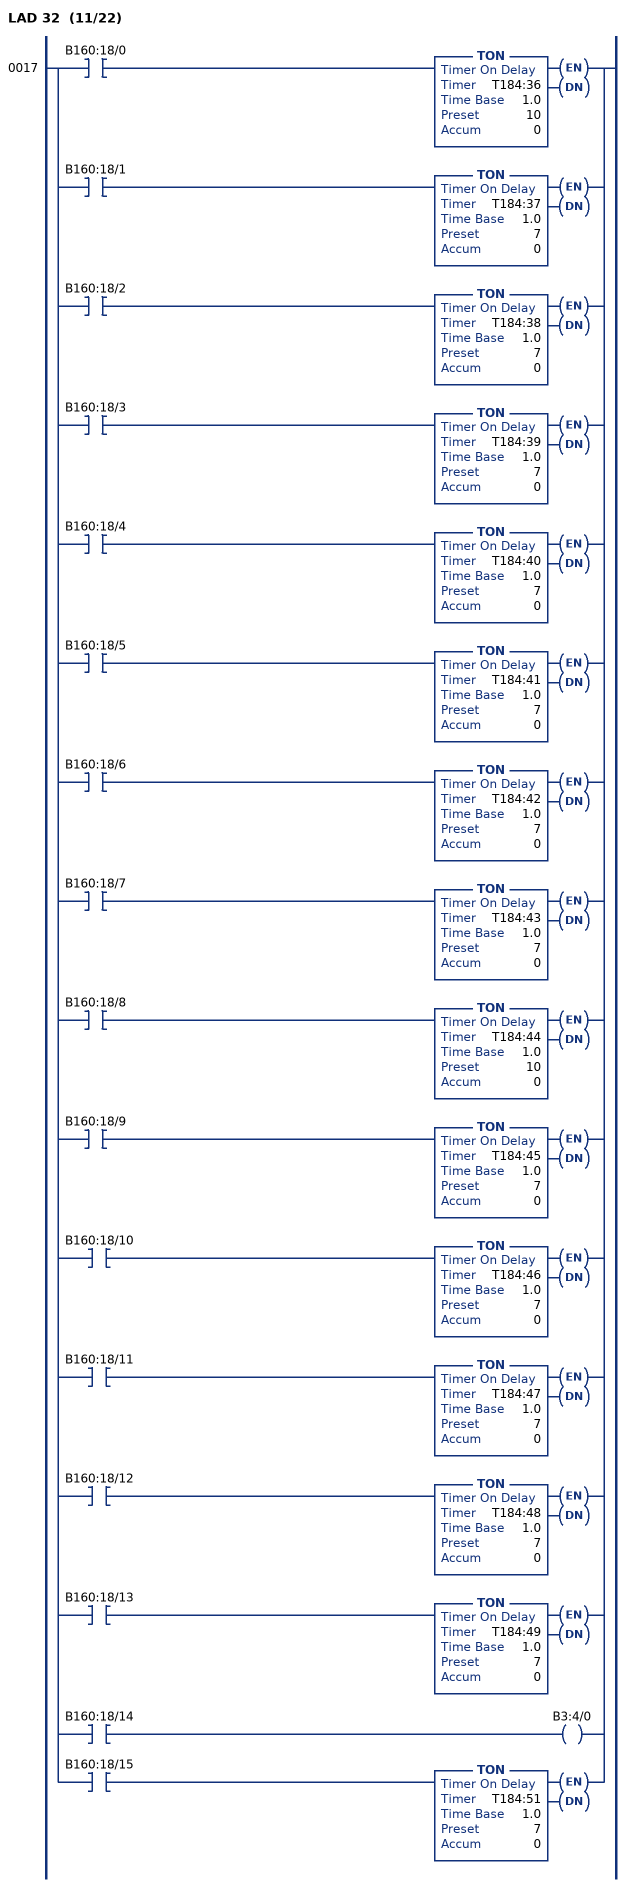
% Rung: 17 %
SOR BST XIC B160:18/0 TON T184:36 1.0 10 0 NXB XIC B160:18/1 TON T184:37 1.0 7 0 NXB XIC B160:18/2 TON T184:38 1.0 7 0 NXB XIC B160:18/3 TON T184:39 1.0 7 0 NXB XIC B160:18/4 TON T184:40 1.0 7 0 NXB XIC B160:18/5 TON T184:41 1.0 7 0 NXB XIC B160:18/6 TON T184:42 1.0 7 0 NXB XIC B160:18/7 TON T184:43 1.0 7 0 NXB XIC B160:18/8 TON T184:44 1.0 10 0 NXB XIC B160:18/9 TON T184:45 1.0 7 0 NXB XIC B160:18/10 TON T184:46 1.0 7 0 NXB XIC B160:18/11 TON T184:47 1.0 7 0 NXB XIC B160:18/12 TON T184:48 1.0 7 0 NXB XIC B160:18/13 TON T184:49 1.0 7 0 NXB XIC B160:18/14 OTE B3:4/0 NXB XIC B160:18/15 TON T184:51 1.0 7 0 BND EOR

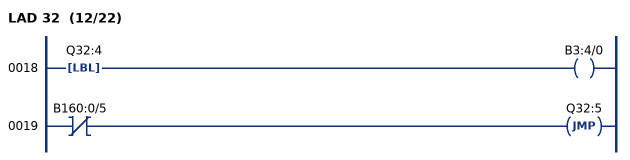
% Rung: 18 %
SOR LBL Q32:4 OTE B3:4/0 EOR
% Rung: 19 %
SOR XIO B160:0/5 JMP Q32:5 EOR

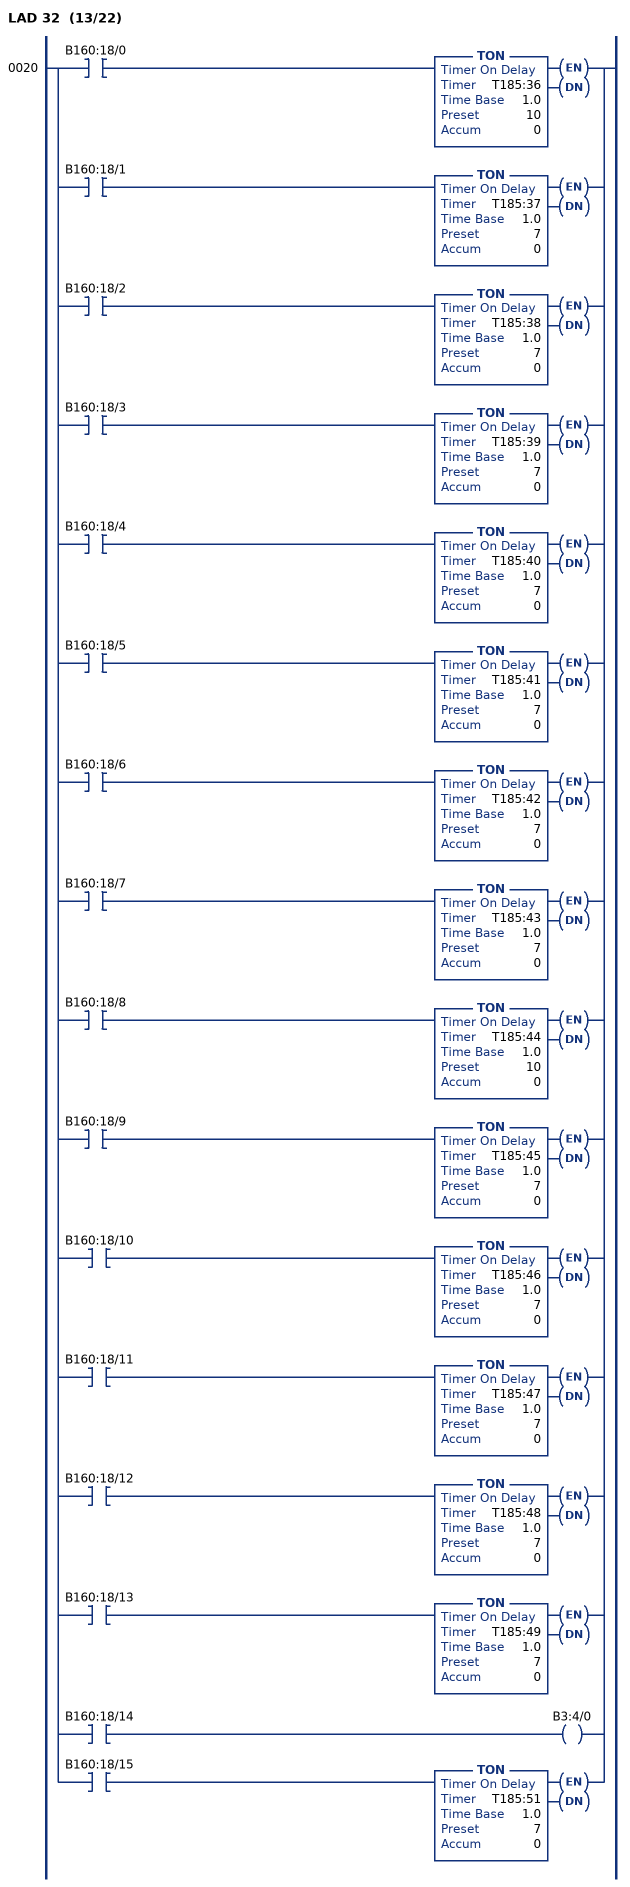
% Rung: 20 %
SOR BST XIC B160:18/0 TON T185:36 1.0 10 0 NXB XIC B160:18/1 TON T185:37 1.0 7 0 NXB XIC B160:18/2 TON T185:38 1.0 7 0 NXB XIC B160:18/3 TON T185:39 1.0 7 0 NXB XIC B160:18/4 TON T185:40 1.0 7 0 NXB XIC B160:18/5 TON T185:41 1.0 7 0 NXB XIC B160:18/6 TON T185:42 1.0 7 0 NXB XIC B160:18/7 TON T185:43 1.0 7 0 NXB XIC B160:18/8 TON T185:44 1.0 10 0 NXB XIC B160:18/9 TON T185:45 1.0 7 0 NXB XIC B160:18/10 TON T185:46 1.0 7 0 NXB XIC B160:18/11 TON T185:47 1.0 7 0 NXB XIC B160:18/12 TON T185:48 1.0 7 0 NXB XIC B160:18/13 TON T185:49 1.0 7 0 NXB XIC B160:18/14 OTE B3:4/0 NXB XIC B160:18/15 TON T185:51 1.0 7 0 BND EOR

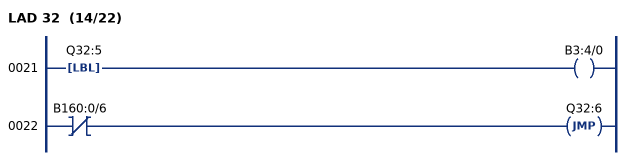
% Rung: 21 %
SOR LBL Q32:5 OTE B3:4/0 EOR
% Rung: 22 %
SOR XIO B160:0/6 JMP Q32:6 EOR

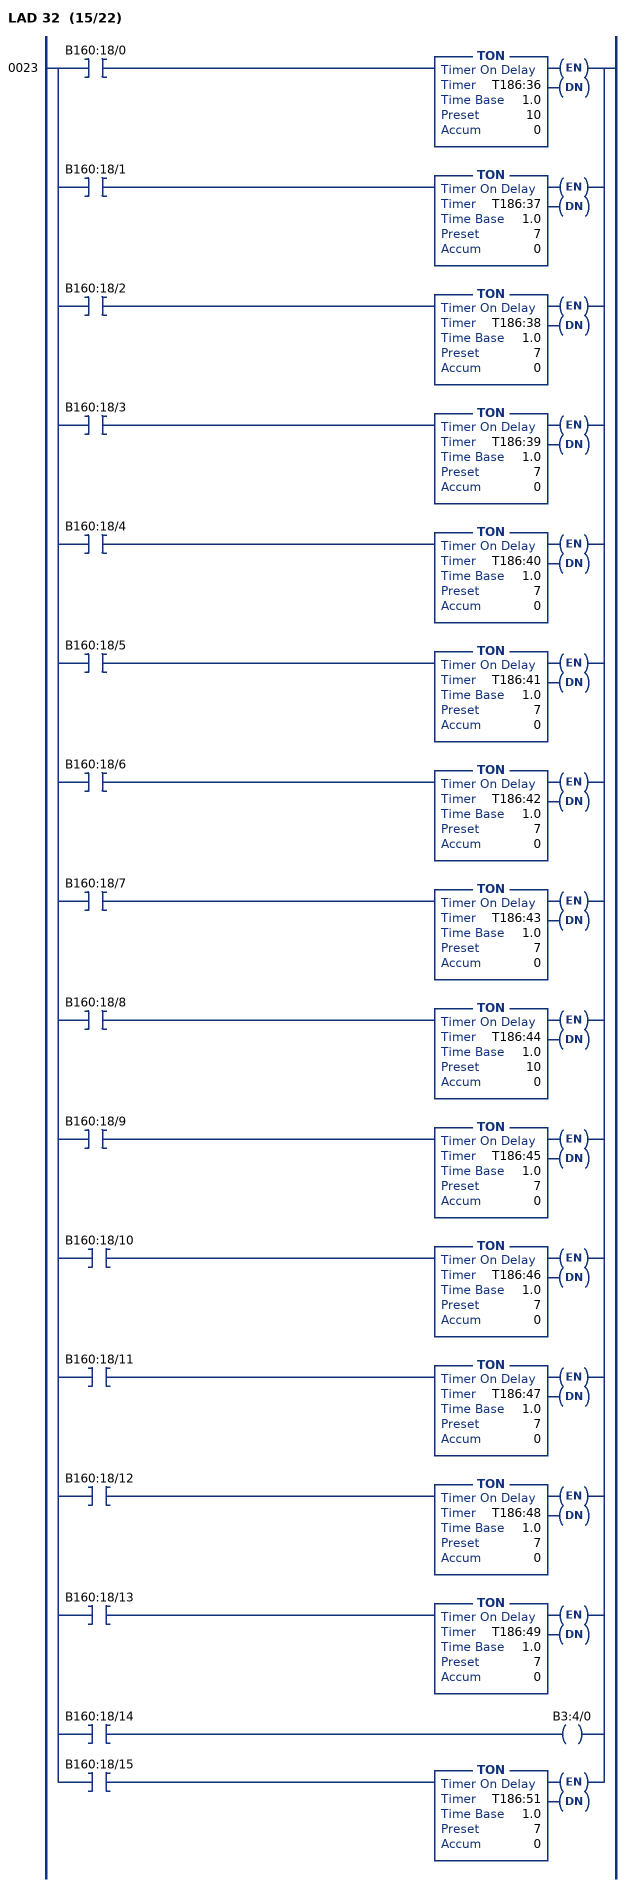
% Rung: 23 %
SOR BST XIC B160:18/0 TON T186:36 1.0 10 0 NXB XIC B160:18/1 TON T186:37 1.0 7 0 NXB XIC B160:18/2 TON T186:38 1.0 7 0 NXB XIC B160:18/3 TON T186:39 1.0 7 0 NXB XIC B160:18/4 TON T186:40 1.0 7 0 NXB XIC B160:18/5 TON T186:41 1.0 7 0 NXB XIC B160:18/6 TON T186:42 1.0 7 0 NXB XIC B160:18/7 TON T186:43 1.0 7 0 NXB XIC B160:18/8 TON T186:44 1.0 10 0 NXB XIC B160:18/9 TON T186:45 1.0 7 0 NXB XIC B160:18/10 TON T186:46 1.0 7 0 NXB XIC B160:18/11 TON T186:47 1.0 7 0 NXB XIC B160:18/12 TON T186:48 1.0 7 0 NXB XIC B160:18/13 TON T186:49 1.0 7 0 NXB XIC B160:18/14 OTE B3:4/0 NXB XIC B160:18/15 TON T186:51 1.0 7 0 BND EOR

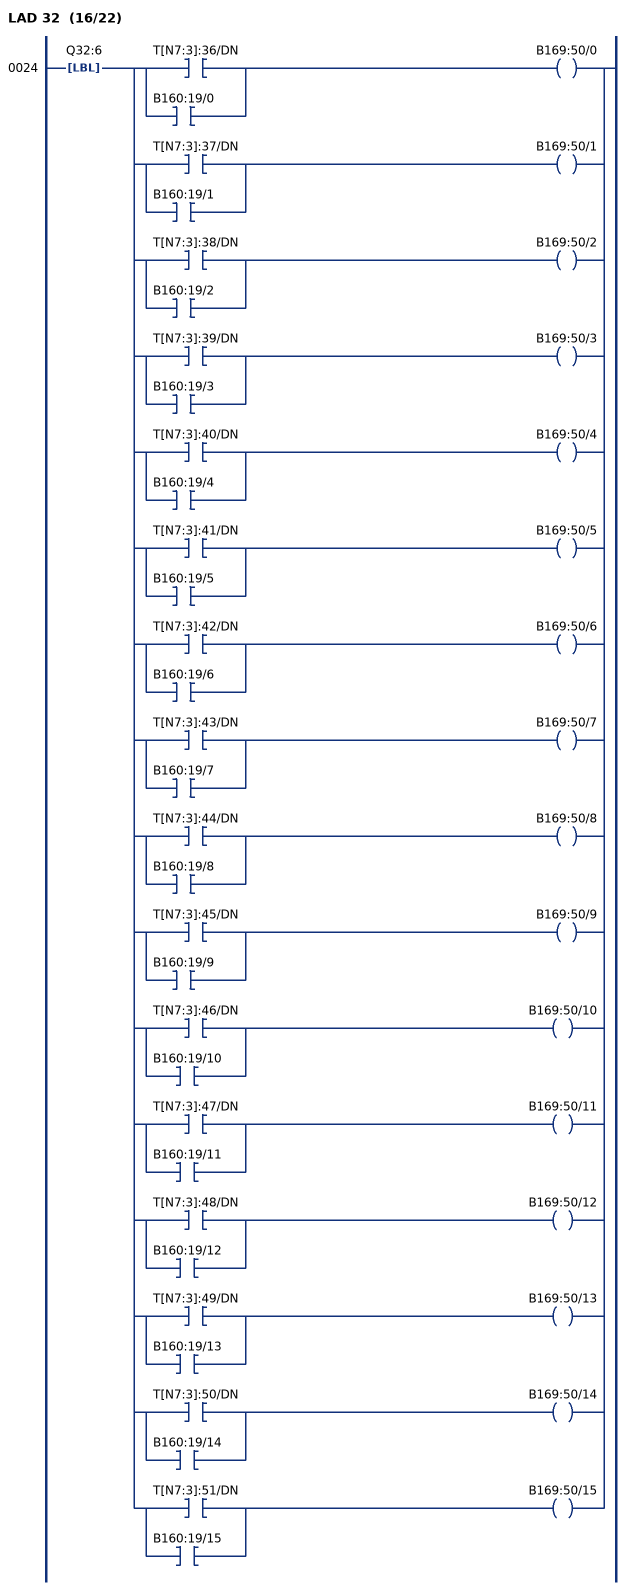
% Rung: 24 %
SOR LBL Q32:6 BST BST XIC T[N7:3]:36/DN NXB XIC B160:19/0 BND OTE B169:50/0 NXB BST XIC T[N7:3]:37/DN NXB XIC B160:19/1 BND OTE B169:50/1 NXB BST XIC T[N7:3]:38/DN NXB XIC B160:19/2 BND OTE B169:50/2 NXB BST XIC T[N7:3]:39/DN NXB XIC B160:19/3 BND OTE B169:50/3 NXB BST XIC T[N7:3]:40/DN NXB XIC B160:19/4 BND OTE B169:50/4 NXB BST XIC T[N7:3]:41/DN NXB XIC B160:19/5 BND OTE B169:50/5 NXB BST XIC T[N7:3]:42/DN NXB XIC B160:19/6 BND OTE B169:50/6 NXB BST XIC T[N7:3]:43/DN NXB XIC B160:19/7 BND OTE B169:50/7 NXB BST XIC T[N7:3]:44/DN NXB XIC B160:19/8 BND OTE B169:50/8 NXB BST XIC T[N7:3]:45/DN NXB XIC B160:19/9 BND OTE B169:50/9 NXB BST XIC T[N7:3]:46/DN NXB XIC B160:19/10 BND OTE B169:50/10 NXB BST XIC T[N7:3]:47/DN NXB XIC B160:19/11 BND OTE B169:50/11 NXB BST XIC T[N7:3]:48/DN NXB XIC B160:19/12 BND OTE B169:50/12 NXB BST XIC T[N7:3]:49/DN NXB XIC B160:19/13 BND OTE B169:50/13 NXB BST XIC T[N7:3]:50/DN NXB XIC B160:19/14 BND OTE B169:50/14 NXB BST XIC T[N7:3]:51/DN NXB XIC B160:19/15 BND OTE B169:50/15 BND EOR

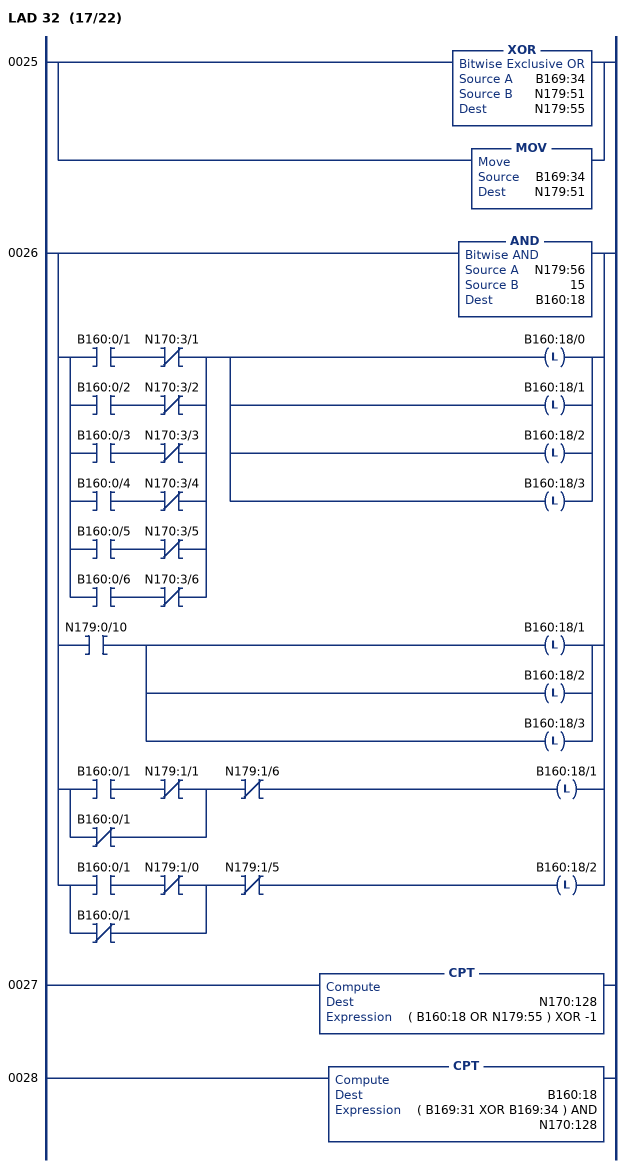
% Rung: 25 %
SOR BST XOR B169:34 N179:51 N179:55 NXB MOV B169:34 N179:51 BND EOR
% Rung: 26 %
SOR BST AND N179:56 15 B160:18 NXB BST XIC B160:0/1 XIO N170:3/1 NXB XIC B160:0/2 XIO N170:3/2 NXB XIC B160:0/3 XIO N170:3/3 NXB XIC B160:0/4 XIO N170:3/4 NXB XIC B160:0/5 XIO N170:3/5 NXB XIC B160:0/6 XIO N170:3/6 BND BST OTL B160:18/0 NXB OTL B160:18/1 NXB OTL B160:18/2 NXB OTL B160:18/3 BND NXB XIC N179:0/10 BST OTL B160:18/1 NXB OTL B160:18/2 NXB OTL B160:18/3 BND NXB BST XIC B160:0/1 XIO N179:1/1 NXB XIO B160:0/1 BND XIO N179:1/6 OTL B160:18/1 NXB BST XIC B160:0/1 XIO N179:1/0 NXB XIO B160:0/1 BND XIO N179:1/5 OTL B160:18/2 BND EOR
% Rung: 27 %
SOR CPT N170:128 " ( B160:18 OR N179:55 ) XOR -1 " EOR
% Rung: 28 %
SOR CPT B160:18 " ( B169:31 XOR B169:34 ) AND N170:128 " EOR

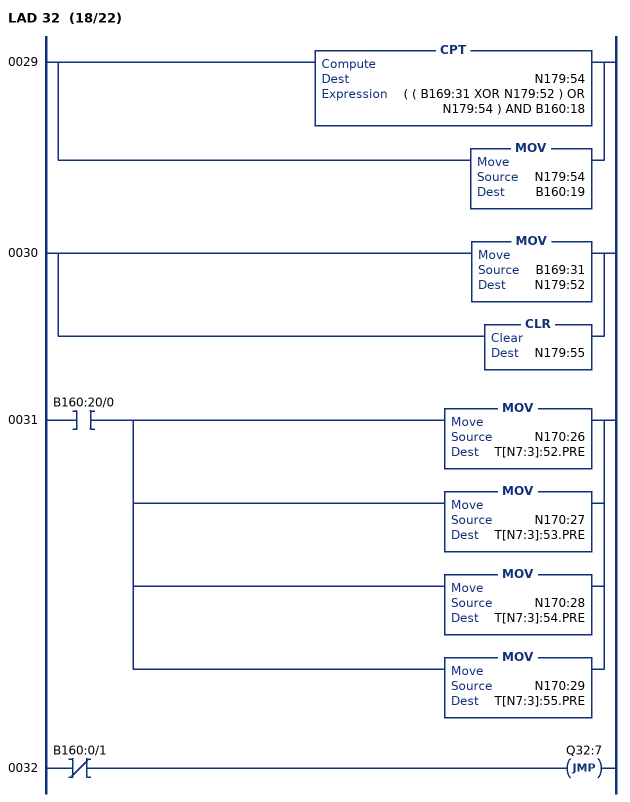
% Rung: 29 %
SOR BST CPT N179:54 " ( ( B169:31 XOR N179:52 ) OR N179:54 ) AND B160:18 " NXB MOV N179:54 B160:19 BND EOR
% Rung: 30 %
SOR BST MOV B169:31 N179:52 NXB CLR N179:55 BND EOR
% Rung: 31 %
SOR XIC B160:20/0 BST MOV N170:26 T[N7:3]:52.PRE NXB MOV N170:27 T[N7:3]:53.PRE NXB MOV N170:28 T[N7:3]:54.PRE NXB MOV N170:29 T[N7:3]:55.PRE BND EOR
% Rung: 32 %
SOR XIO B160:0/1 JMP Q32:7 EOR

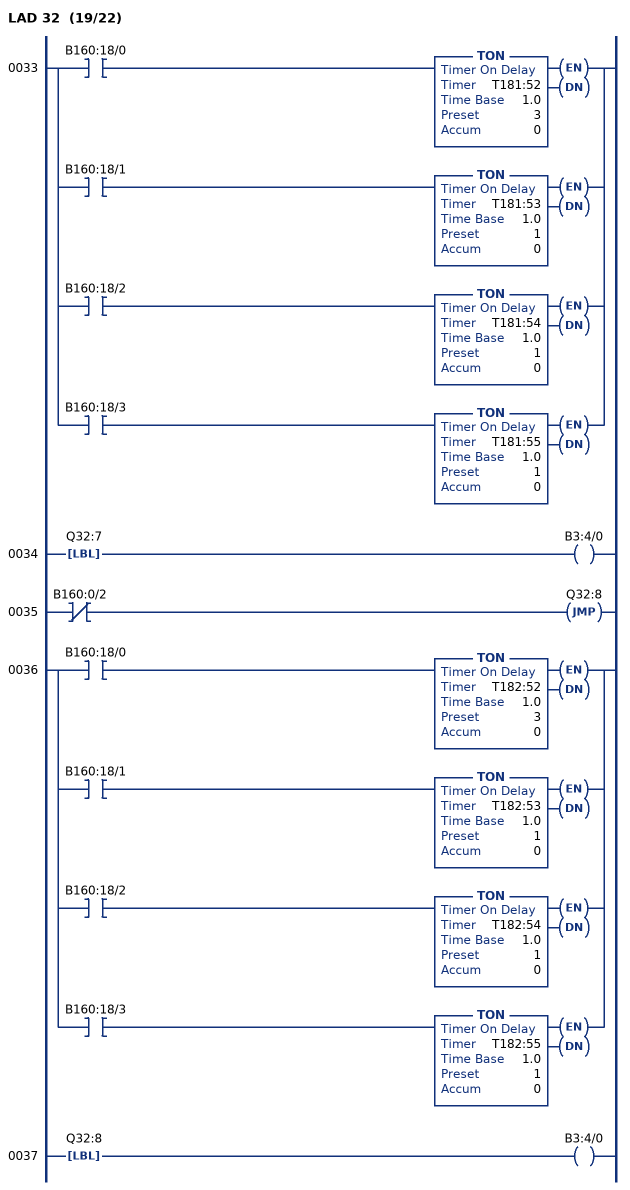
% Rung: 33 %
SOR BST XIC B160:18/0 TON T181:52 1.0 3 0 NXB XIC B160:18/1 TON T181:53 1.0 1 0 NXB XIC B160:18/2 TON T181:54 1.0 1 0 NXB XIC B160:18/3 TON T181:55 1.0 1 0 BND EOR
% Rung: 34 %
SOR LBL Q32:7 OTE B3:4/0 EOR
% Rung: 35 %
SOR XIO B160:0/2 JMP Q32:8 EOR
% Rung: 36 %
SOR BST XIC B160:18/0 TON T182:52 1.0 3 0 NXB XIC B160:18/1 TON T182:53 1.0 1 0 NXB XIC B160:18/2 TON T182:54 1.0 1 0 NXB XIC B160:18/3 TON T182:55 1.0 1 0 BND EOR
% Rung: 37 %
SOR LBL Q32:8 OTE B3:4/0 EOR

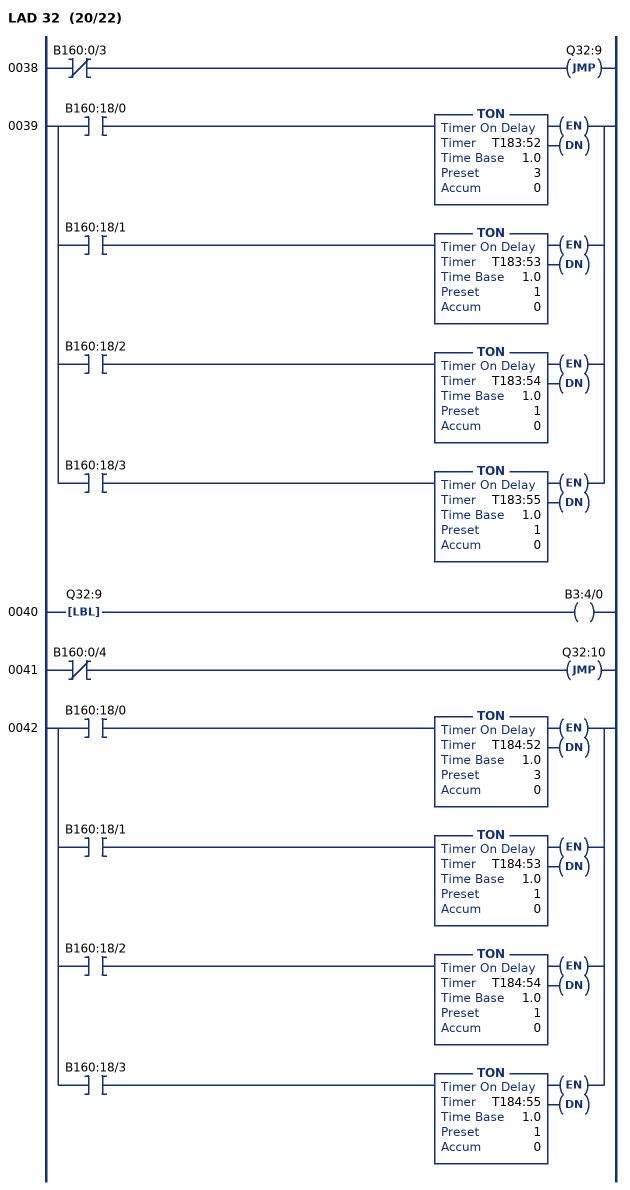
% Rung: 38 %
SOR XIO B160:0/3 JMP Q32:9 EOR
% Rung: 39 %
SOR BST XIC B160:18/0 TON T183:52 1.0 3 0 NXB XIC B160:18/1 TON T183:53 1.0 1 0 NXB XIC B160:18/2 TON T183:54 1.0 1 0 NXB XIC B160:18/3 TON T183:55 1.0 1 0 BND EOR
% Rung: 40 %
SOR LBL Q32:9 OTE B3:4/0 EOR
% Rung: 41 %
SOR XIO B160:0/4 JMP Q32:10 EOR
% Rung: 42 %
SOR BST XIC B160:18/0 TON T184:52 1.0 3 0 NXB XIC B160:18/1 TON T184:53 1.0 1 0 NXB XIC B160:18/2 TON T184:54 1.0 1 0 NXB XIC B160:18/3 TON T184:55 1.0 1 0 BND EOR

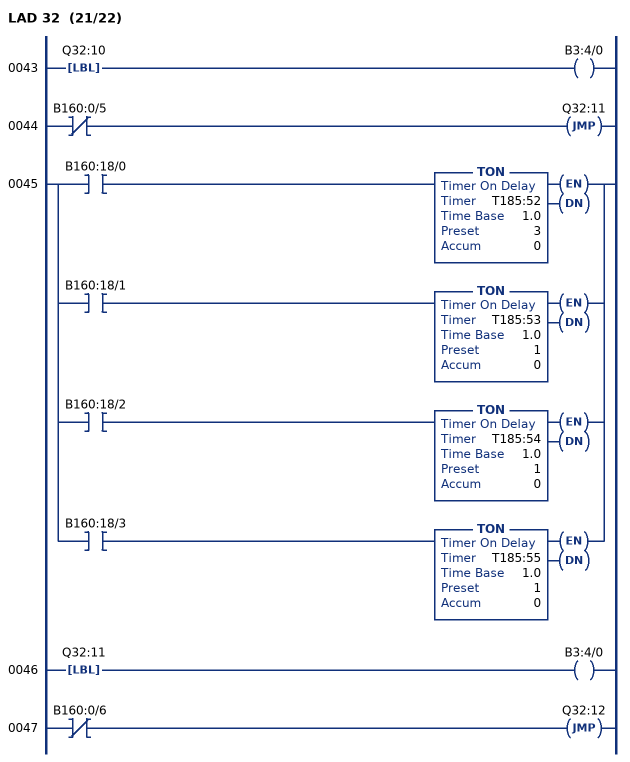
% Rung: 43 %
SOR LBL Q32:10 OTE B3:4/0 EOR
% Rung: 44 %
SOR XIO B160:0/5 JMP Q32:11 EOR
% Rung: 45 %
SOR BST XIC B160:18/0 TON T185:52 1.0 3 0 NXB XIC B160:18/1 TON T185:53 1.0 1 0 NXB XIC B160:18/2 TON T185:54 1.0 1 0 NXB XIC B160:18/3 TON T185:55 1.0 1 0 BND EOR
% Rung: 46 %
SOR LBL Q32:11 OTE B3:4/0 EOR
% Rung: 47 %
SOR XIO B160:0/6 JMP Q32:12 EOR

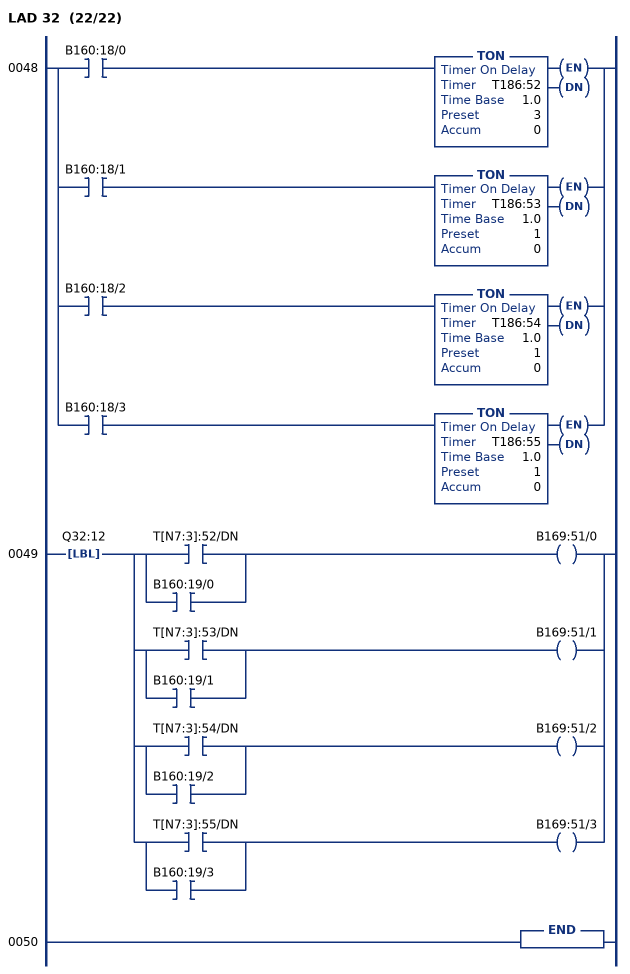
% Rung: 48 %
SOR BST XIC B160:18/0 TON T186:52 1.0 3 0 NXB XIC B160:18/1 TON T186:53 1.0 1 0 NXB XIC B160:18/2 TON T186:54 1.0 1 0 NXB XIC B160:18/3 TON T186:55 1.0 1 0 BND EOR
% Rung: 49 %
SOR LBL Q32:12 BST BST XIC T[N7:3]:52/DN NXB XIC B160:19/0 BND OTE B169:51/0 NXB BST XIC T[N7:3]:53/DN NXB XIC B160:19/1 BND OTE B169:51/1 NXB BST XIC T[N7:3]:54/DN NXB XIC B160:19/2 BND OTE B169:51/2 NXB BST XIC T[N7:3]:55/DN NXB XIC B160:19/3 BND OTE B169:51/3 BND EOR
% Rung: 50 %
SOR END EOR

LADDER 33
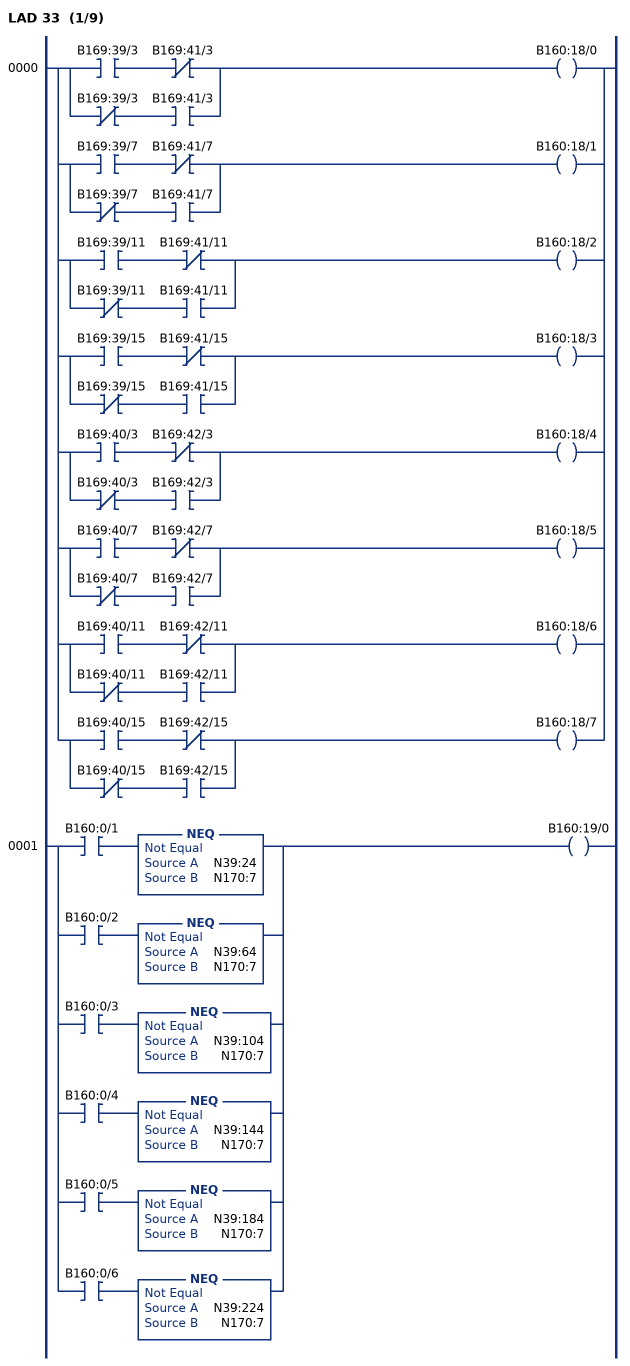
% Rung: 0 %
SOR BST BST XIC B169:39/3 XIO B169:41/3 NXB XIO B169:39/3 XIC B169:41/3 BND OTE B160:18/0 NXB BST XIC B169:39/7 XIO B169:41/7 NXB XIO B169:39/7 XIC B169:41/7 BND OTE B160:18/1 NXB BST XIC B169:39/11 XIO B169:41/11 NXB XIO B169:39/11 XIC B169:41/11 BND OTE B160:18/2 NXB BST XIC B169:39/15 XIO B169:41/15 NXB XIO B169:39/15 XIC B169:41/15 BND OTE B160:18/3 NXB BST XIC B169:40/3 XIO B169:42/3 NXB XIO B169:40/3 XIC B169:42/3 BND OTE B160:18/4 NXB BST XIC B169:40/7 XIO B169:42/7 NXB XIO B169:40/7 XIC B169:42/7 BND OTE B160:18/5 NXB BST XIC B169:40/11 XIO B169:42/11 NXB XIO B169:40/11 XIC B169:42/11 BND OTE B160:18/6 NXB BST XIC B169:40/15 XIO B169:42/15 NXB XIO B169:40/15 XIC B169:42/15 BND OTE B160:18/7 BND EOR
% Rung: 1 %
SOR BST XIC B160:0/1 NEQ N39:24 N170:7 NXB XIC B160:0/2 NEQ N39:64 N170:7 NXB XIC B160:0/3 NEQ N39:104 N170:7 NXB XIC B160:0/4 NEQ N39:144 N170:7 NXB XIC B160:0/5 NEQ N39:184 N170:7 NXB XIC B160:0/6 NEQ N39:224 N170:7 BND OTE B160:19/0 EOR

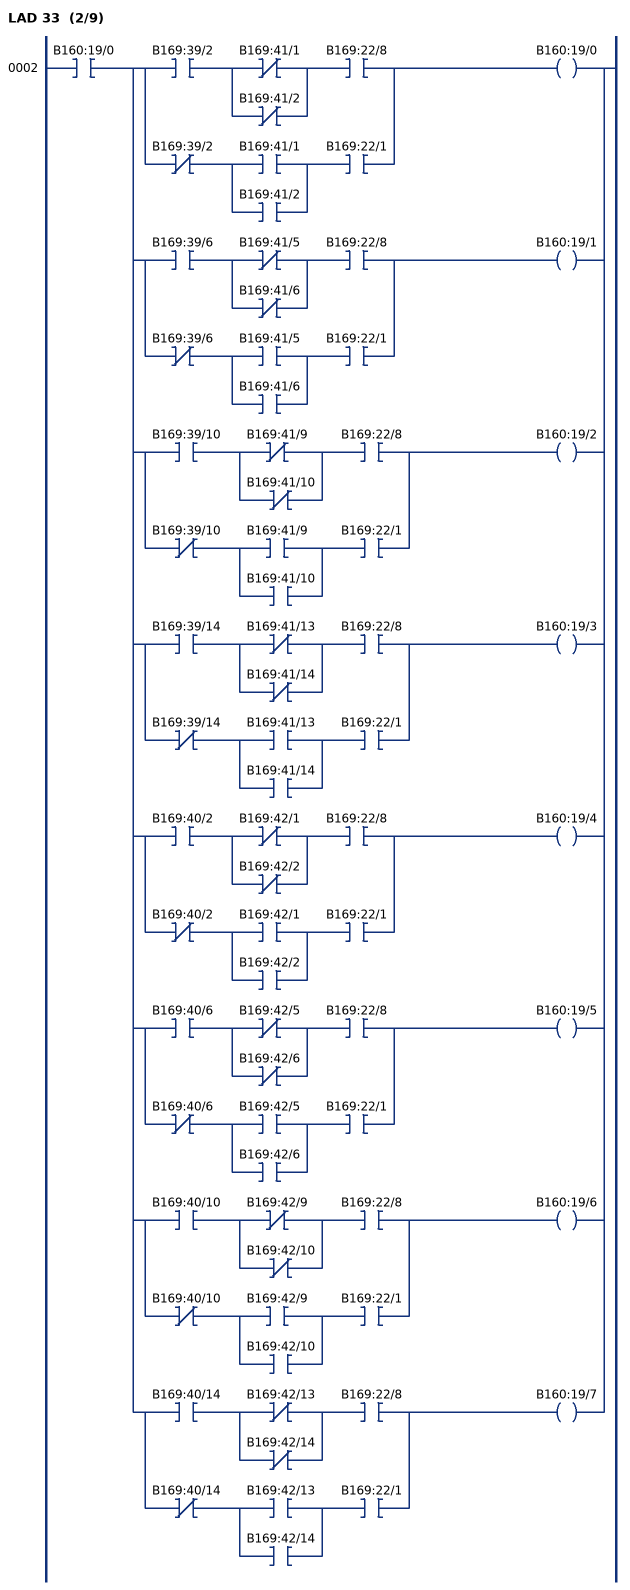
% Rung: 2 %
SOR XIC B160:19/0 BST BST XIC B169:39/2 BST XIO B169:41/1 NXB XIO B169:41/2 BND XIC B169:22/8 NXB XIO B169:39/2 BST XIC B169:41/1 NXB XIC B169:41/2 BND XIC B169:22/1 BND OTE B160:19/0 NXB BST XIC B169:39/6 BST XIO B169:41/5 NXB XIO B169:41/6 BND XIC B169:22/8 NXB XIO B169:39/6 BST XIC B169:41/5 NXB XIC B169:41/6 BND XIC B169:22/1 BND OTE B160:19/1 NXB BST XIC B169:39/10 BST XIO B169:41/9 NXB XIO B169:41/10 BND XIC B169:22/8 NXB XIO B169:39/10 BST XIC B169:41/9 NXB XIC B169:41/10 BND XIC B169:22/1 BND OTE B160:19/2 NXB BST XIC B169:39/14 BST XIO B169:41/13 NXB XIO B169:41/14 BND XIC B169:22/8 NXB XIO B169:39/14 BST XIC B169:41/13 NXB XIC B169:41/14 BND XIC B169:22/1 BND OTE B160:19/3 NXB BST XIC B169:40/2 BST XIO B169:42/1 NXB XIO B169:42/2 BND XIC B169:22/8 NXB XIO B169:40/2 BST XIC B169:42/1 NXB XIC B169:42/2 BND XIC B169:22/1 BND OTE B160:19/4 NXB BST XIC B169:40/6 BST XIO B169:42/5 NXB XIO B169:42/6 BND XIC B169:22/8 NXB XIO B169:40/6 BST XIC B169:42/5 NXB XIC B169:42/6 BND XIC B169:22/1 BND OTE B160:19/5 NXB BST XIC B169:40/10 BST XIO B169:42/9 NXB XIO B169:42/10 BND XIC B169:22/8 NXB XIO B169:40/10 BST XIC B169:42/9 NXB XIC B169:42/10 BND XIC B169:22/1 BND OTE B160:19/6 NXB BST XIC B169:40/14 BST XIO B169:42/13 NXB XIO B169:42/14 BND XIC B169:22/8 NXB XIO B169:40/14 BST XIC B169:42/13 NXB XIC B169:42/14 BND XIC B169:22/1 BND OTE B160:19/7 BND EOR

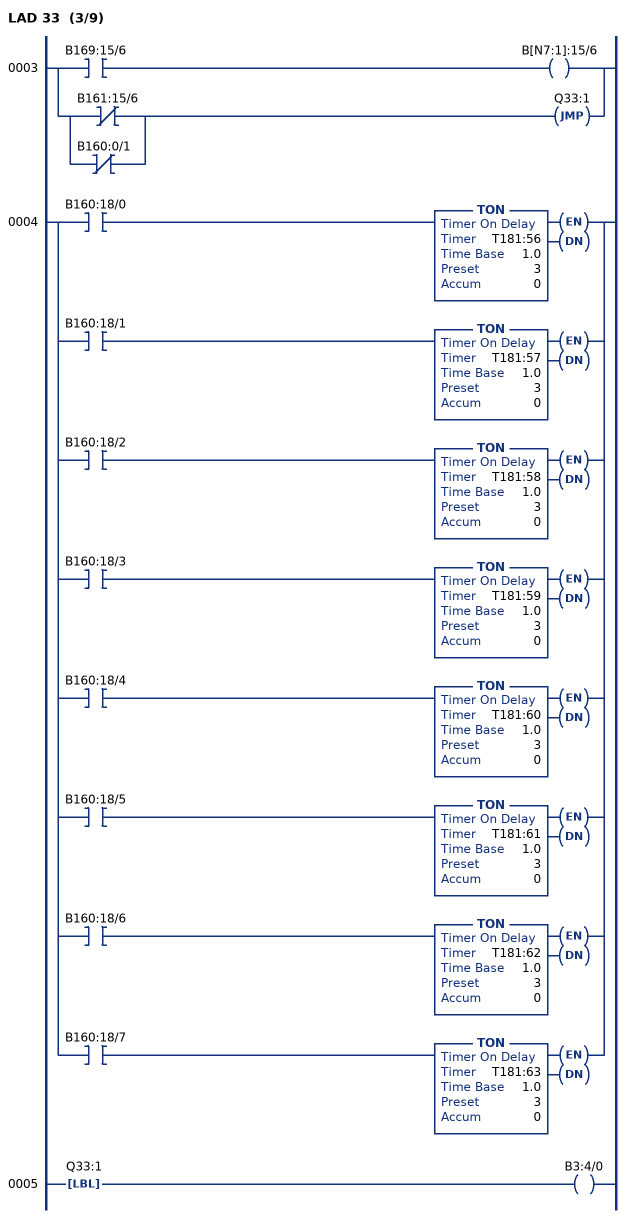
% Rung: 3 %
SOR BST XIC B169:15/6 OTE B[N7:1]:15/6 NXB BST XIO B161:15/6 NXB XIO B160:0/1 BND JMP Q33:1 BND EOR
% Rung: 4 %
SOR BST XIC B160:18/0 TON T181:56 1.0 3 0 NXB XIC B160:18/1 TON T181:57 1.0 3 0 NXB XIC B160:18/2 TON T181:58 1.0 3 0 NXB XIC B160:18/3 TON T181:59 1.0 3 0 NXB XIC B160:18/4 TON T181:60 1.0 3 0 NXB XIC B160:18/5 TON T181:61 1.0 3 0 NXB XIC B160:18/6 TON T181:62 1.0 3 0 NXB XIC B160:18/7 TON T181:63 1.0 3 0 BND EOR
% Rung: 5 %
SOR LBL Q33:1 OTE B3:4/0 EOR

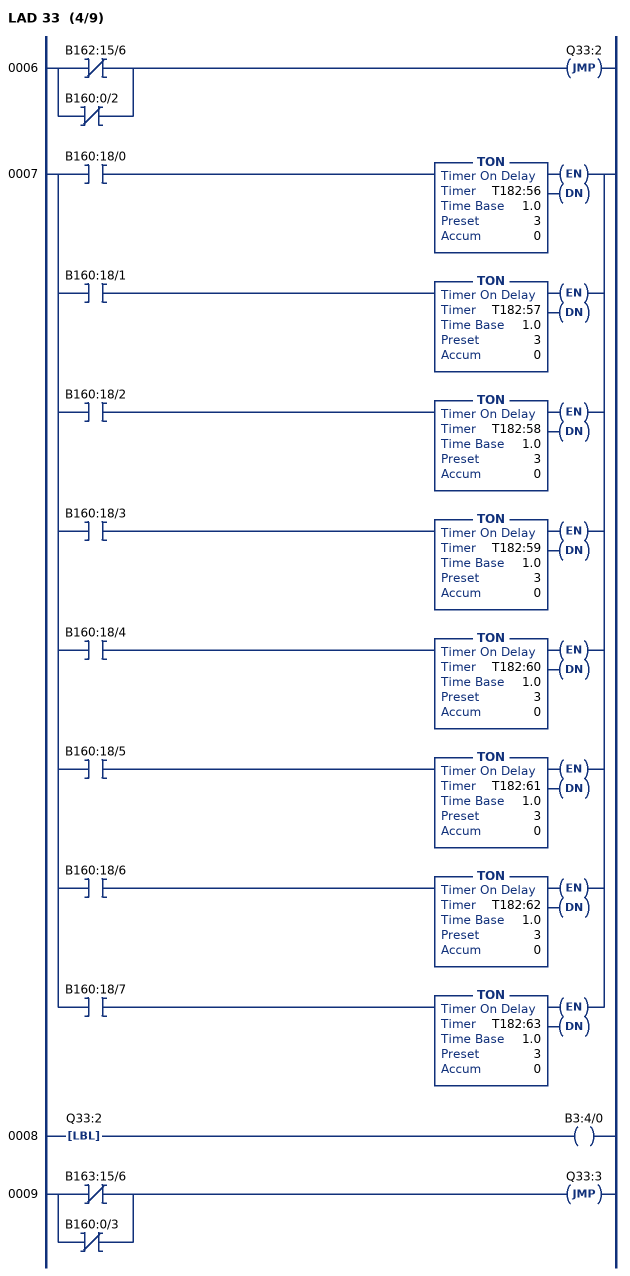
% Rung: 6 %
SOR BST XIO B162:15/6 NXB XIO B160:0/2 BND JMP Q33:2 EOR
% Rung: 7 %
SOR BST XIC B160:18/0 TON T182:56 1.0 3 0 NXB XIC B160:18/1 TON T182:57 1.0 3 0 NXB XIC B160:18/2 TON T182:58 1.0 3 0 NXB XIC B160:18/3 TON T182:59 1.0 3 0 NXB XIC B160:18/4 TON T182:60 1.0 3 0 NXB XIC B160:18/5 TON T182:61 1.0 3 0 NXB XIC B160:18/6 TON T182:62 1.0 3 0 NXB XIC B160:18/7 TON T182:63 1.0 3 0 BND EOR
% Rung: 8 %
SOR LBL Q33:2 OTE B3:4/0 EOR
% Rung: 9 %
SOR BST XIO B163:15/6 NXB XIO B160:0/3 BND JMP Q33:3 EOR

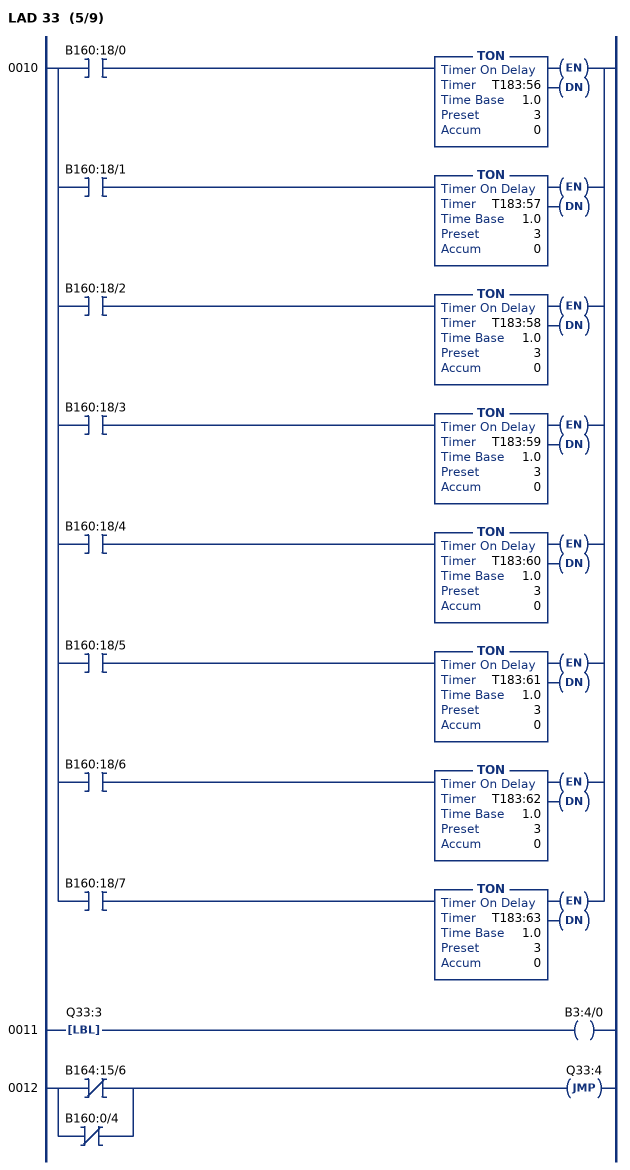
% Rung: 10 %
SOR BST XIC B160:18/0 TON T183:56 1.0 3 0 NXB XIC B160:18/1 TON T183:57 1.0 3 0 NXB XIC B160:18/2 TON T183:58 1.0 3 0 NXB XIC B160:18/3 TON T183:59 1.0 3 0 NXB XIC B160:18/4 TON T183:60 1.0 3 0 NXB XIC B160:18/5 TON T183:61 1.0 3 0 NXB XIC B160:18/6 TON T183:62 1.0 3 0 NXB XIC B160:18/7 TON T183:63 1.0 3 0 BND EOR
% Rung: 11 %
SOR LBL Q33:3 OTE B3:4/0 EOR
% Rung: 12 %
SOR BST XIO B164:15/6 NXB XIO B160:0/4 BND JMP Q33:4 EOR

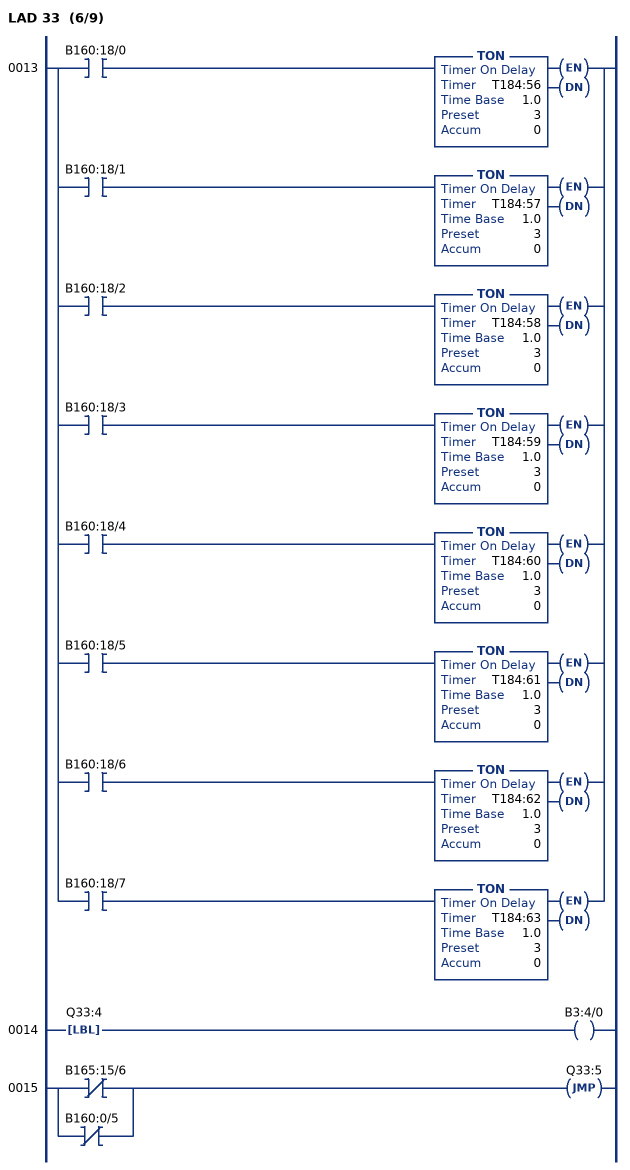
% Rung: 13 %
SOR BST XIC B160:18/0 TON T184:56 1.0 3 0 NXB XIC B160:18/1 TON T184:57 1.0 3 0 NXB XIC B160:18/2 TON T184:58 1.0 3 0 NXB XIC B160:18/3 TON T184:59 1.0 3 0 NXB XIC B160:18/4 TON T184:60 1.0 3 0 NXB XIC B160:18/5 TON T184:61 1.0 3 0 NXB XIC B160:18/6 TON T184:62 1.0 3 0 NXB XIC B160:18/7 TON T184:63 1.0 3 0 BND EOR
% Rung: 14 %
SOR LBL Q33:4 OTE B3:4/0 EOR
% Rung: 15 %
SOR BST XIO B165:15/6 NXB XIO B160:0/5 BND JMP Q33:5 EOR

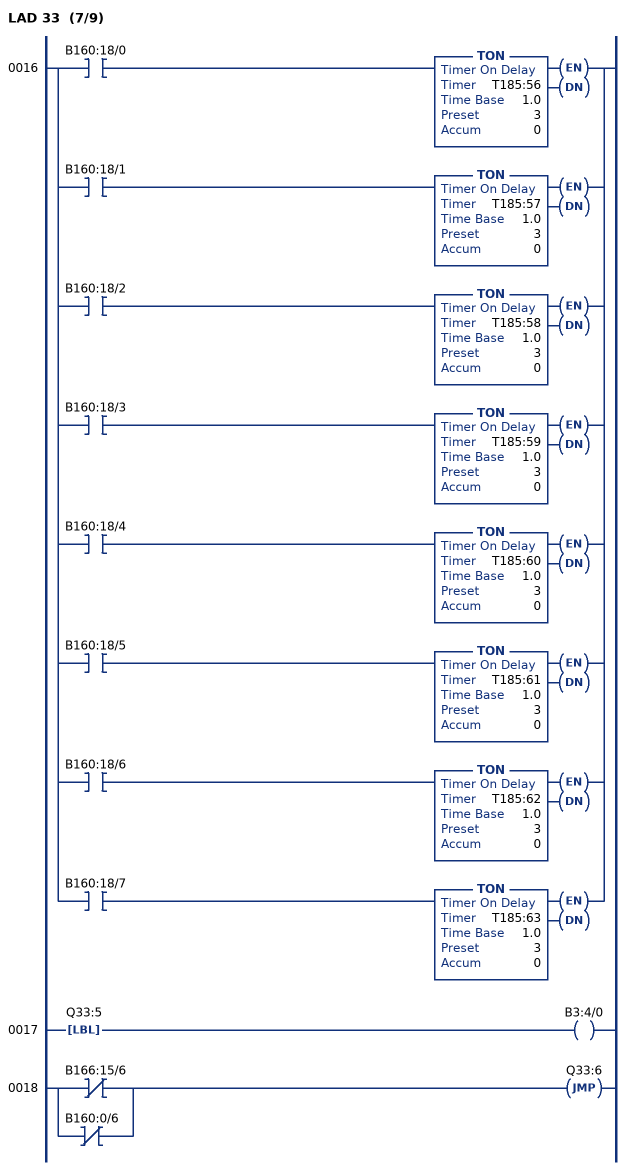
% Rung: 16 %
SOR BST XIC B160:18/0 TON T185:56 1.0 3 0 NXB XIC B160:18/1 TON T185:57 1.0 3 0 NXB XIC B160:18/2 TON T185:58 1.0 3 0 NXB XIC B160:18/3 TON T185:59 1.0 3 0 NXB XIC B160:18/4 TON T185:60 1.0 3 0 NXB XIC B160:18/5 TON T185:61 1.0 3 0 NXB XIC B160:18/6 TON T185:62 1.0 3 0 NXB XIC B160:18/7 TON T185:63 1.0 3 0 BND EOR
% Rung: 17 %
SOR LBL Q33:5 OTE B3:4/0 EOR
% Rung: 18 %
SOR BST XIO B166:15/6 NXB XIO B160:0/6 BND JMP Q33:6 EOR

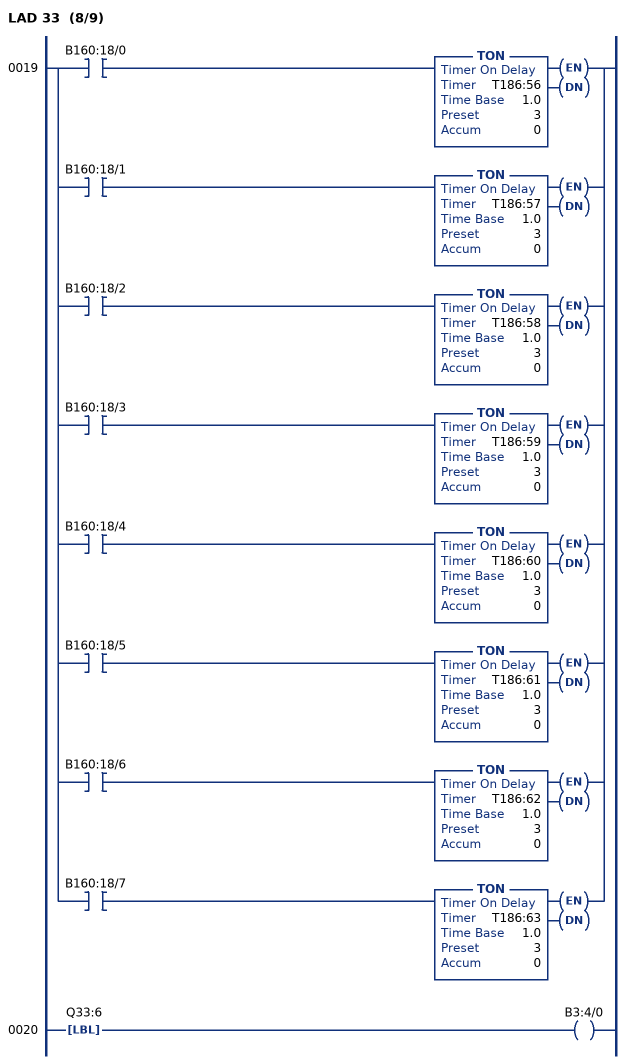
% Rung: 19 %
SOR BST XIC B160:18/0 TON T186:56 1.0 3 0 NXB XIC B160:18/1 TON T186:57 1.0 3 0 NXB XIC B160:18/2 TON T186:58 1.0 3 0 NXB XIC B160:18/3 TON T186:59 1.0 3 0 NXB XIC B160:18/4 TON T186:60 1.0 3 0 NXB XIC B160:18/5 TON T186:61 1.0 3 0 NXB XIC B160:18/6 TON T186:62 1.0 3 0 NXB XIC B160:18/7 TON T186:63 1.0 3 0 BND EOR
% Rung: 20 %
SOR LBL Q33:6 OTE B3:4/0 EOR

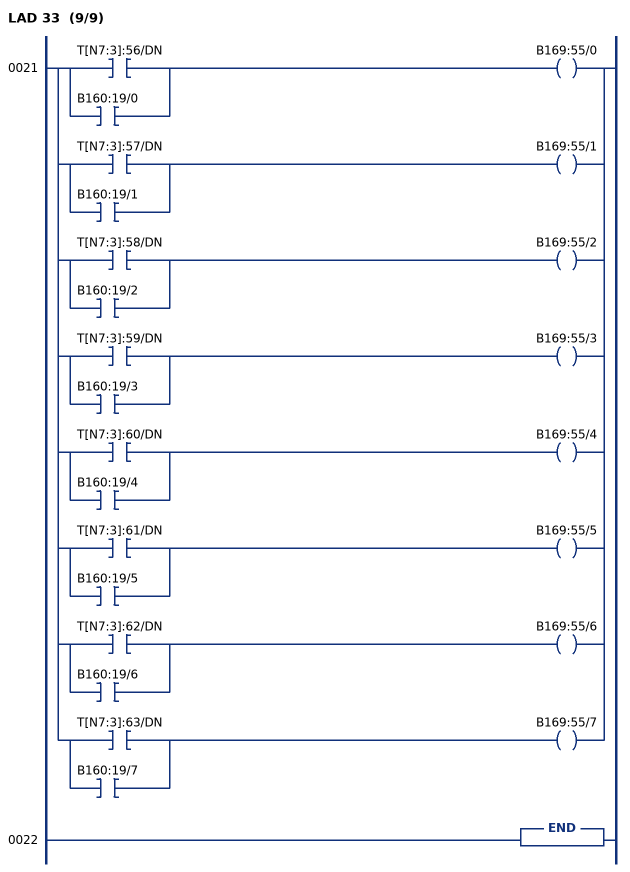
% Rung: 21 %
SOR BST BST XIC T[N7:3]:56/DN NXB XIC B160:19/0 BND OTE B169:55/0 NXB BST XIC T[N7:3]:57/DN NXB XIC B160:19/1 BND OTE B169:55/1 NXB BST XIC T[N7:3]:58/DN NXB XIC B160:19/2 BND OTE B169:55/2 NXB BST XIC T[N7:3]:59/DN NXB XIC B160:19/3 BND OTE B169:55/3 NXB BST XIC T[N7:3]:60/DN NXB XIC B160:19/4 BND OTE B169:55/4 NXB BST XIC T[N7:3]:61/DN NXB XIC B160:19/5 BND OTE B169:55/5 NXB BST XIC T[N7:3]:62/DN NXB XIC B160:19/6 BND OTE B169:55/6 NXB BST XIC T[N7:3]:63/DN NXB XIC B160:19/7 BND OTE B169:55/7 BND EOR
% Rung: 22 %
SOR END EOR

LADDER 37
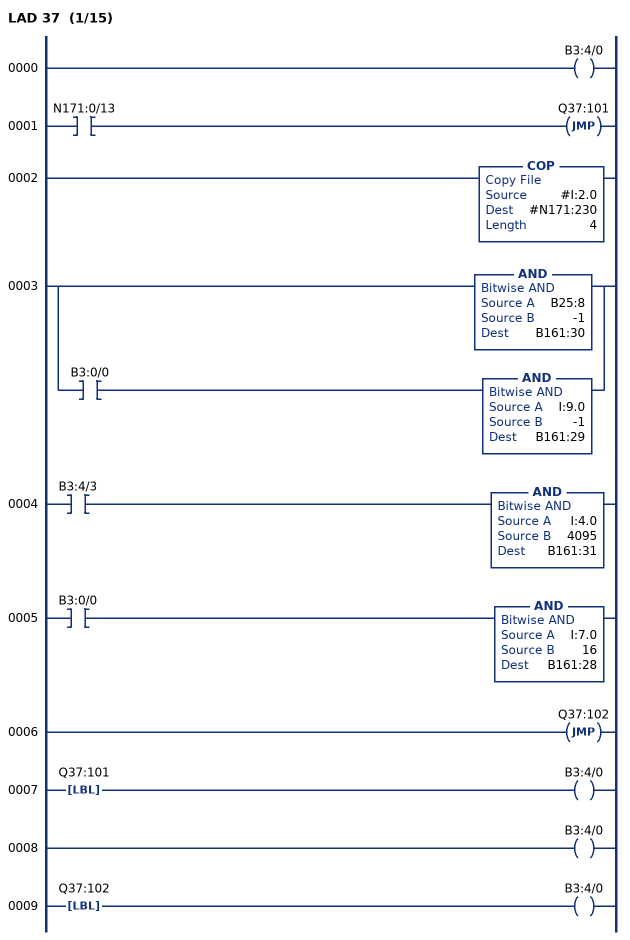
% Rung: 0 %
SOR OTE B3:4/0 EOR
% Rung: 1 %
SOR XIC N171:0/13 JMP Q37:101 EOR
% Rung: 2 %
SOR COP #I:2.0 #N171:230 4 EOR
% Rung: 3 %
SOR BST AND B25:8 -1 B161:30 NXB XIC B3:0/0 AND I:9.0 -1 B161:29 BND EOR
% Rung: 4 %
SOR XIC B3:4/3 AND I:4.0 4095 B161:31 EOR
% Rung: 5 %
SOR XIC B3:0/0 AND I:7.0 16 B161:28 EOR
% Rung: 6 %
SOR JMP Q37:102 EOR
% Rung: 7 %
SOR LBL Q37:101 OTE B3:4/0 EOR
% Rung: 8 %
SOR OTE B3:4/0 EOR
% Rung: 9 %
SOR LBL Q37:102 OTE B3:4/0 EOR

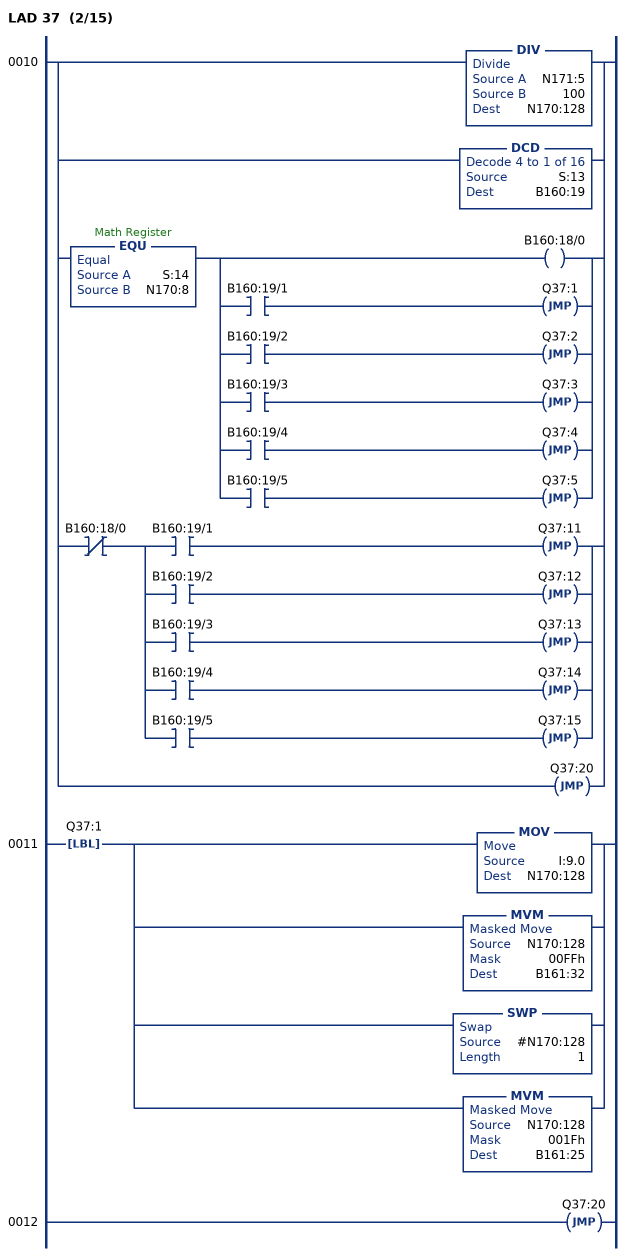
% Rung: 10 %
SOR BST DIV N171:5 100 N170:128 NXB DCD S:13 B160:19 NXB EQU S:14 N170:8 BST OTE B160:18/0 NXB XIC B160:19/1 JMP Q37:1 NXB XIC B160:19/2 JMP Q37:2 NXB XIC B160:19/3 JMP Q37:3 NXB XIC B160:19/4 JMP Q37:4 NXB XIC B160:19/5 JMP Q37:5 BND NXB XIO B160:18/0 BST XIC B160:19/1 JMP Q37:11 NXB XIC B160:19/2 JMP Q37:12 NXB XIC B160:19/3 JMP Q37:13 NXB XIC B160:19/4 JMP Q37:14 NXB XIC B160:19/5 JMP Q37:15 BND NXB JMP Q37:20 BND EOR
%   S:13  "Math Register" %
%   S:14  "Math Register" %
% Rung: 11 %
SOR LBL Q37:1 BST MOV I:9.0 N170:128 NXB MVM N170:128 00FFh B161:32 NXB SWP #N170:128 1 NXB MVM N170:128 001Fh B161:25 BND EOR
% Rung: 12 %
SOR JMP Q37:20 EOR

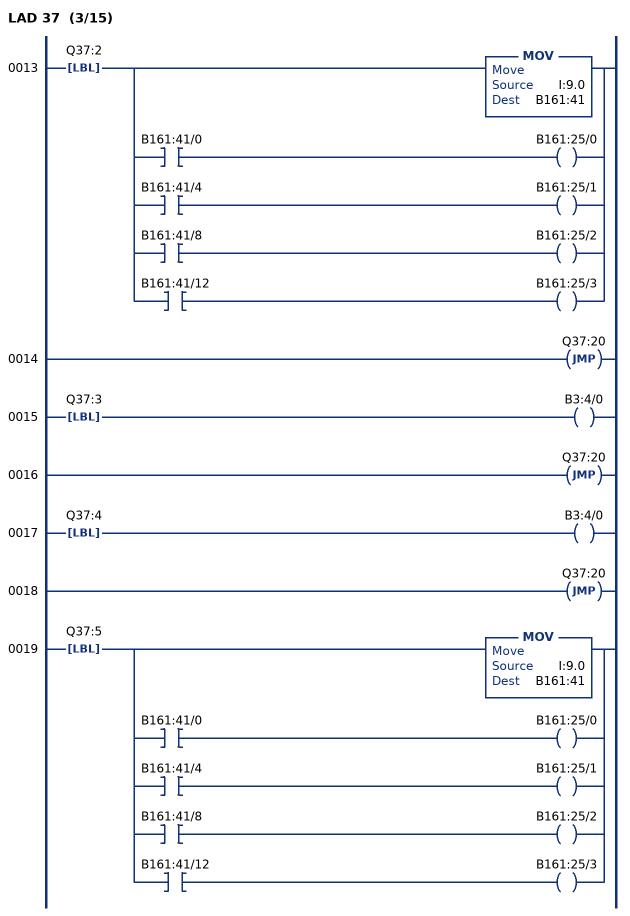
% Rung: 13 %
SOR LBL Q37:2 BST MOV I:9.0 B161:41 NXB XIC B161:41/0 OTE B161:25/0 NXB XIC B161:41/4 OTE B161:25/1 NXB XIC B161:41/8 OTE B161:25/2 NXB XIC B161:41/12 OTE B161:25/3 BND EOR
% Rung: 14 %
SOR JMP Q37:20 EOR
% Rung: 15 %
SOR LBL Q37:3 OTE B3:4/0 EOR
% Rung: 16 %
SOR JMP Q37:20 EOR
% Rung: 17 %
SOR LBL Q37:4 OTE B3:4/0 EOR
% Rung: 18 %
SOR JMP Q37:20 EOR
% Rung: 19 %
SOR LBL Q37:5 BST MOV I:9.0 B161:41 NXB XIC B161:41/0 OTE B161:25/0 NXB XIC B161:41/4 OTE B161:25/1 NXB XIC B161:41/8 OTE B161:25/2 NXB XIC B161:41/12 OTE B161:25/3 BND EOR

